{attribute 'GeneratedUsingTerminal: EL2034-0000-0018'}
{attribute addProperty BoxType "EL2034-0000-0018"}
{attribute addProperty Id "OutputAT %Q*BOOL1"}
{attribute addProperty CRC "1120571895"}
{attribute addProperty Size "1"}
TYPE Channel_42CA91F7 EXTENDS OutputBase_10CEE7DE :
STRUCT
	{attribute addProperty Name "Output"}
	Output AT %Q* : BOOL;
END_STRUCT
END_TYPE

(* stored: Version 1.2.0.0, ProductVersion 3.1.4024.11
   DUT Channel_42CA91F7: Id {34c1be56-0c3b-4cf5-8284-37b7fe804b00} *)
